FUNCTION_BLOCK minimum
VAR_INPUT
	x: ARRAY[0..399] OF LREAL;
END_VAR
VAR_OUTPUT
	ex: LREAL;
	idx: DINT;
END_VAR
VAR
	k: DINT;
	tmp: LREAL;
END_VAR


ex := x[0];
idx := 1;

FOR k := 0 TO 398 DO 
    tmp := x[k + 1];

    IF ex > tmp THEN 
        ex := tmp;
        idx := k + 2;
    END_IF;

END_FOR;

END_FUNCTION_BLOCK

(* stored: Version 1.1.0.1, ProductVersion 3.1.4024.11
   POU minimum: Id {f1f80bee-f2e8-4509-aa8a-3c33f46826f3}, SpecialFunc None *)
